DATA_BLOCK "G279M"
TITLE =DBG279M  HEATING KILN 1 + 2
//COPYRIGHT:    (C) 2009  BUHLER AG, CH-9240 UZWIL, SWITZERLAND
//
//PRODUCT:      WinCoS_BIW01_09
//
//TITLE:        HEATING KILN 1 + 2
//                Machine group DB
//                Maschinengruppen-DB
//
//-------------------------------------------------------------------------
//
//IDENT:        AUTHOR:             DEPT:             DATE:
//
//P01_DB379.1.0 K.Renz              CSB41             30.Sep.2009
//              1st Release
//
//-------------------------------------------------------------------------
//
//PURPOSE:
//
//MANUAL :
//
//RESTRICTIONS:
//
//-------------------------------------------------------------------------
AUTHOR : KR
FAMILY : USW
NAME : DBG279M
VERSION : 0.0

"G279M_Code"
BEGIN
   Gr.FcCode := 0;
   Gr.Spare2 := 0;
   Gr.Spare4 := 0;
   Gr.Spare6 := 0;
   Gr.OutEmptyingTime := 0;
   Gr.ChangeBit.spare := B#16#0;
   Gr.ChangeBit.CBit1 := FALSE;
   Gr.ChangeBit.CBit2 := FALSE;
   Gr.ChangeBit.CBit3 := FALSE;
   Gr.ChangeBit.CBit4 := FALSE;
   Gr.StCode := 0;
   Gr.InEnableGr := FALSE;
   Gr.CmdContinue := FALSE;
   Gr.CmdRestartIdling := FALSE;
   Gr.InReleaseEmptyingTime := FALSE;
   Gr.InFeeding := FALSE;
   Gr.InOutAutostartMan := FALSE;
   Gr.InPreStart := FALSE;
   Gr.CmdManualOff := FALSE;
   Gr.CmdOff := FALSE;
   Gr.CmdOn := FALSE;
   Gr.CmdNext := FALSE;
   Gr.CmdFaultReset := FALSE;
   Gr.InOccupied := FALSE;
   Gr.InManual := FALSE;
   Gr.InLoadedSec := FALSE;
   Gr.InSeqStop := FALSE;
   Gr.ModePassive := FALSE;
   Gr.ModeActive := FALSE;
   Gr.ModeIdling := FALSE;
   Gr.spare163 := FALSE;
   Gr.spare164 := FALSE;
   Gr.spare165 := FALSE;
   Gr.spare166 := FALSE;
   Gr.spare167 := FALSE;
   Gr.StStopped := FALSE;
   Gr.StStarting := FALSE;
   Gr.StStarted := FALSE;
   Gr.StStopping := FALSE;
   Gr.StFault := FALSE;
   Gr.OutLoaded := FALSE;
   Gr.OutWarning := FALSE;
   Gr.OutFeeding := FALSE;
   Gr.OutEnableEl := FALSE;
   Gr.OutEnable1 := FALSE;
   Gr.OutHWStop := FALSE;
   Gr.OutDPFault := FALSE;
   Gr.OutAutostart := FALSE;
   Gr.OutManual := FALSE;
   Gr.OutHornOn := FALSE;
   Gr.OutEnablePrevGr := FALSE;
   Gr.VarStopped := FALSE;
   Gr.VarStarted := FALSE;
   Gr.VarFault := FALSE;
   Gr.VarStartwarning := FALSE;
   Gr.VarFlag1s := FALSE;
   Gr.OutEmptyingTimeDone := FALSE;
   Gr.OutNewWay := FALSE;
   Gr.OutSeqStop := FALSE;
   Gr.OutIdlingTime := 0;
   Gr.InCodePreselect := 0;
   Gr.InLine := 0;
   Gr.InCode := 0;
   Gr.OutCode := 0;
   Gr.Par.ParObjectNo := 27900;
   Gr.Par.ParMgr := TRUE;
   Gr.Par.ParWgr := FALSE;
   Gr.Par.ParGgr := FALSE;
   Gr.Par.ParHornCode := 10;
   Gr.Par.ParIdling := 2;
   Gr.Par.ParEmptyingTime := 0;
   Gr.Par.Para1_0 := FALSE;
   Gr.Par.Para1_1 := FALSE;
   Gr.Par.Para1_2 := FALSE;
   Gr.Par.Para1_3 := FALSE;
   Gr.Par.Para1_4 := FALSE;
   Gr.Par.Para1_5 := FALSE;
   Gr.Par.Para1_6 := FALSE;
   Gr.Par.Para1_7 := FALSE;
   Gr.Par.Para1_8 := FALSE;
   Gr.Par.Para1_9 := FALSE;
   Gr.Par.Para1_10 := FALSE;
   Gr.Par.Para1_11 := FALSE;
   Gr.Par.Para1_12 := FALSE;
   Gr.Par.Para1_13 := FALSE;
   Gr.Par.Para1_14 := FALSE;
   Gr.Par.Para1_15 := FALSE;
   Gr.Par.Para2 := 0;
   Gr.Par.Para3 := 0;
   Gr.Par.Para4 := 0;
   Gr.Par.Para5 := 0;
   InOutValue1 := L#0;
   InOutValue2 := L#0;
   OutWayConflict := FALSE;
   OutSelectionOk := FALSE;
   CmdNewValue := FALSE;
   CmdNewJob := FALSE;
   OutCodeOK := FALSE;
   InEndOfJob := FALSE;
   staWayOk := FALSE;
   EdgeStartRelease := FALSE;
   USW8 := FALSE;
   USW9 := FALSE;
   USW10 := FALSE;
   _A_3191_BTE10_Active := FALSE;
   _A_3291_BTE10_Active := FALSE;
   USW13 := FALSE;
   USW14 := FALSE;
   USW15 := FALSE;
   A_3161_KCL11.StCode := 0;
   A_3161_KCL11.InMonTrue := FALSE;
   A_3161_KCL11.InMonFalse := FALSE;
   A_3161_KCL11.InPreAlarmTrue := FALSE;
   A_3161_KCL11.InPreAlarmFalse := FALSE;
   A_3161_KCL11.InStopTrueTime := FALSE;
   A_3161_KCL11.InStopFalseTime := FALSE;
   A_3161_KCL11.InpTrue := FALSE;
   A_3161_KCL11.InpFaultDev := FALSE;
   A_3161_KCL11.CmdRstTrueTime := FALSE;
   A_3161_KCL11.CmdRstFalseTime := FALSE;
   A_3161_KCL11.CmdRunTimeoutTime := FALSE;
   A_3161_KCL11.CmdFaultReset := FALSE;
   A_3161_KCL11.InLocal := FALSE;
   A_3161_KCL11.spare0305 := FALSE;
   A_3161_KCL11.InReport := FALSE;
   A_3161_KCL11.OutTimeoutTime := FALSE;
   A_3161_KCL11.InHWStop := FALSE;
   A_3161_KCL11.InDPFault := FALSE;
   A_3161_KCL11.OutPreAlarmTrue := FALSE;
   A_3161_KCL11.OutPreAlarmFalse := FALSE;
   A_3161_KCL11.OutFlagPos := FALSE;
   A_3161_KCL11.OutFlagNeg := FALSE;
   A_3161_KCL11.OutpFaultReset := FALSE;
   A_3161_KCL11.OutTrue := FALSE;
   A_3161_KCL11.StFalse := FALSE;
   A_3161_KCL11.StCtoTrue := FALSE;
   A_3161_KCL11.StTrue := FALSE;
   A_3161_KCL11.StCtoFalse := FALSE;
   A_3161_KCL11.StFault := FALSE;
   A_3161_KCL11.OutAlarmNrLog := 0;
   A_3161_KCL11.Par.ParObjectNo := 27901;
   A_3161_KCL11.Par.ParMsgType := 7154;
   A_3161_KCL11.Par.ParHornCode := 10;
   A_3161_KCL11.Par.ParLogOff := FALSE;
   A_3161_KCL11.Par.spare0401 := FALSE;
   A_3161_KCL11.Par.Par2WorkingCond := FALSE;
   A_3161_KCL11.Par.ParFaultRetry := FALSE;
   A_3161_KCL11.Par.ParBinLevel := FALSE;
   A_3161_KCL11.Par.ParDelayChange := 20;
   A_3161_KCL11.Par.ParDelayTrue := 10;
   A_3161_KCL11.Par.ParDelayFalse := 0;
   A_3161_KCL11.Par.ParTimeoutTrue := 0;
   A_3161_KCL11.Par.ParTimeoutFalse := 0;
   A_3161_KCL11.Par.OutMonTime := 0;
   A_3161_KCL11.Par.OutTransitionTime := 0;
   A_3161_KCL11.Par.OutMonTrue := FALSE;
   A_3161_KCL11.Par.OutMonFalse := FALSE;
   A_3161_KCL11.Par.OutFlagFaultDev := FALSE;
   A_3161_KCL11.Par.OutDelayTime := 0;
   A_3161_KCL11_EXT_ON.StCode := 0;
   A_3161_KCL11_EXT_ON.InEnable := FALSE;
   A_3161_KCL11_EXT_ON.spare0201 := FALSE;
   A_3161_KCL11_EXT_ON.InContinuous := FALSE;
   A_3161_KCL11_EXT_ON.spare0203 := FALSE;
   A_3161_KCL11_EXT_ON.spare0204 := FALSE;
   A_3161_KCL11_EXT_ON.spare0205 := FALSE;
   A_3161_KCL11_EXT_ON.InpRun := FALSE;
   A_3161_KCL11_EXT_ON.InpFaultDev := FALSE;
   A_3161_KCL11_EXT_ON.CmdOff := FALSE;
   A_3161_KCL11_EXT_ON.CmdOn := FALSE;
   A_3161_KCL11_EXT_ON.CmdNext := FALSE;
   A_3161_KCL11_EXT_ON.CmdFaultReset := FALSE;
   A_3161_KCL11_EXT_ON.InLocal := FALSE;
   A_3161_KCL11_EXT_ON.InManual := FALSE;
   A_3161_KCL11_EXT_ON.InReport := FALSE;
   A_3161_KCL11_EXT_ON.InSeqStop := FALSE;
   A_3161_KCL11_EXT_ON.InHWStop := FALSE;
   A_3161_KCL11_EXT_ON.InDPFault := FALSE;
   A_3161_KCL11_EXT_ON.OutIdling := FALSE;
   A_3161_KCL11_EXT_ON.OutWarning := FALSE;
   A_3161_KCL11_EXT_ON.spare0404 := FALSE;
   A_3161_KCL11_EXT_ON.spare0405 := FALSE;
   A_3161_KCL11_EXT_ON.OutpFaultReset := FALSE;
   A_3161_KCL11_EXT_ON.OutpRun := FALSE;
   A_3161_KCL11_EXT_ON.StStopped := FALSE;
   A_3161_KCL11_EXT_ON.StStarting := FALSE;
   A_3161_KCL11_EXT_ON.StStarted := FALSE;
   A_3161_KCL11_EXT_ON.spare0503 := FALSE;
   A_3161_KCL11_EXT_ON.StFault := FALSE;
   A_3161_KCL11_EXT_ON.StFalse := FALSE;
   A_3161_KCL11_EXT_ON.spare0506 := FALSE;
   A_3161_KCL11_EXT_ON.OutPausing := FALSE;
   A_3161_KCL11_EXT_ON.OutAlarmNrLog := 0;
   A_3161_KCL11_EXT_ON.Par.ParObjectNo := 27902;
   A_3161_KCL11_EXT_ON.Par.ParMsgType := 7002;
   A_3161_KCL11_EXT_ON.Par.ParHornCode := 0;
   A_3161_KCL11_EXT_ON.Par.ParLogOff := FALSE;
   A_3161_KCL11_EXT_ON.Par.ParManual := TRUE;
   A_3161_KCL11_EXT_ON.Par.ParContinuous := TRUE;
   A_3161_KCL11_EXT_ON.Par.ParPulse := FALSE;
   A_3161_KCL11_EXT_ON.Par.ParPulsing := FALSE;
   A_3161_KCL11_EXT_ON.Par.ParFilter := FALSE;
   A_3161_KCL11_EXT_ON.Par.ParOnTime := 10;
   A_3161_KCL11_EXT_ON.Par.ParOffTime := 0;
   A_3161_KCL11_EXT_ON.Par.ParIdlingTime := 0;
   A_3161_KCL11_EXT_ON.Par.ParDelayTime := 0;
   A_3161_KCL11_EXT_ON.Par.OutTime := 0;
   A_3161_KCL11_EXT_ON.Par.OutDelayTime := 0;
   A_3161_KCL11_EXT_ON.Par.spare26 := 0;
   A_3161_KCL11_EXT_ON.Par.spare28 := 0;
   A_3161_KCL11_EXT_ON.Par.InOutManPulseLen := 0;
   A_3161_KCL11_ON.StCode := 0;
   A_3161_KCL11_ON.InMonTrue := FALSE;
   A_3161_KCL11_ON.InMonFalse := FALSE;
   A_3161_KCL11_ON.InPreAlarmTrue := FALSE;
   A_3161_KCL11_ON.InPreAlarmFalse := FALSE;
   A_3161_KCL11_ON.InStopTrueTime := FALSE;
   A_3161_KCL11_ON.InStopFalseTime := FALSE;
   A_3161_KCL11_ON.InpTrue := FALSE;
   A_3161_KCL11_ON.InpFaultDev := FALSE;
   A_3161_KCL11_ON.CmdRstTrueTime := FALSE;
   A_3161_KCL11_ON.CmdRstFalseTime := FALSE;
   A_3161_KCL11_ON.CmdRunTimeoutTime := FALSE;
   A_3161_KCL11_ON.CmdFaultReset := FALSE;
   A_3161_KCL11_ON.InLocal := FALSE;
   A_3161_KCL11_ON.spare0305 := FALSE;
   A_3161_KCL11_ON.InReport := FALSE;
   A_3161_KCL11_ON.OutTimeoutTime := FALSE;
   A_3161_KCL11_ON.InHWStop := FALSE;
   A_3161_KCL11_ON.InDPFault := FALSE;
   A_3161_KCL11_ON.OutPreAlarmTrue := FALSE;
   A_3161_KCL11_ON.OutPreAlarmFalse := FALSE;
   A_3161_KCL11_ON.OutFlagPos := FALSE;
   A_3161_KCL11_ON.OutFlagNeg := FALSE;
   A_3161_KCL11_ON.OutpFaultReset := FALSE;
   A_3161_KCL11_ON.OutTrue := FALSE;
   A_3161_KCL11_ON.StFalse := FALSE;
   A_3161_KCL11_ON.StCtoTrue := FALSE;
   A_3161_KCL11_ON.StTrue := FALSE;
   A_3161_KCL11_ON.StCtoFalse := FALSE;
   A_3161_KCL11_ON.StFault := FALSE;
   A_3161_KCL11_ON.OutAlarmNrLog := 0;
   A_3161_KCL11_ON.Par.ParObjectNo := 27903;
   A_3161_KCL11_ON.Par.ParMsgType := 7154;
   A_3161_KCL11_ON.Par.ParHornCode := 0;
   A_3161_KCL11_ON.Par.ParLogOff := FALSE;
   A_3161_KCL11_ON.Par.spare0401 := FALSE;
   A_3161_KCL11_ON.Par.Par2WorkingCond := FALSE;
   A_3161_KCL11_ON.Par.ParFaultRetry := FALSE;
   A_3161_KCL11_ON.Par.ParBinLevel := FALSE;
   A_3161_KCL11_ON.Par.ParDelayChange := 20;
   A_3161_KCL11_ON.Par.ParDelayTrue := 10;
   A_3161_KCL11_ON.Par.ParDelayFalse := 0;
   A_3161_KCL11_ON.Par.ParTimeoutTrue := 0;
   A_3161_KCL11_ON.Par.ParTimeoutFalse := 0;
   A_3161_KCL11_ON.Par.OutMonTime := 0;
   A_3161_KCL11_ON.Par.OutTransitionTime := 0;
   A_3161_KCL11_ON.Par.OutMonTrue := FALSE;
   A_3161_KCL11_ON.Par.OutMonFalse := FALSE;
   A_3161_KCL11_ON.Par.OutFlagFaultDev := FALSE;
   A_3161_KCL11_ON.Par.OutDelayTime := 0;
   A_3161_KCL11_AI.StCode := 0;
   A_3161_KCL11_AI.InMonLL := FALSE;
   A_3161_KCL11_AI.InMonL := FALSE;
   A_3161_KCL11_AI.InMonMid := FALSE;
   A_3161_KCL11_AI.InMonH := FALSE;
   A_3161_KCL11_AI.InMonHH := FALSE;
   A_3161_KCL11_AI.spare0205 := FALSE;
   A_3161_KCL11_AI.InpFaultAI := FALSE;
   A_3161_KCL11_AI.InpFaultDev := FALSE;
   A_3161_KCL11_AI.InHWStop := FALSE;
   A_3161_KCL11_AI.InDPFault := FALSE;
   A_3161_KCL11_AI.InDisable := FALSE;
   A_3161_KCL11_AI.CmdFaultReset := FALSE;
   A_3161_KCL11_AI.InLocal := FALSE;
   A_3161_KCL11_AI.spare0305 := FALSE;
   A_3161_KCL11_AI.InReport := FALSE;
   A_3161_KCL11_AI.spare0307 := FALSE;
   A_3161_KCL11_AI.OutLL := FALSE;
   A_3161_KCL11_AI.OutL := FALSE;
   A_3161_KCL11_AI.OutH := FALSE;
   A_3161_KCL11_AI.OutHH := FALSE;
   A_3161_KCL11_AI.OutOverflow := FALSE;
   A_3161_KCL11_AI.spare0405 := FALSE;
   A_3161_KCL11_AI.OutFaultAI := FALSE;
   A_3161_KCL11_AI.spare0407 := FALSE;
   A_3161_KCL11_AI.StLL := FALSE;
   A_3161_KCL11_AI.StL := FALSE;
   A_3161_KCL11_AI.StMid := FALSE;
   A_3161_KCL11_AI.StH := FALSE;
   A_3161_KCL11_AI.StHH := FALSE;
   A_3161_KCL11_AI.StFaultAI := FALSE;
   A_3161_KCL11_AI.OutWarning := FALSE;
   A_3161_KCL11_AI.OutFaulted := FALSE;
   A_3161_KCL11_AI.InpValue := 0;
   A_3161_KCL11_AI.OutValuePc := 0;
   A_3161_KCL11_AI.OutValueUnits := L#0;
   A_3161_KCL11_AI.Msg.WarningDoneLL := FALSE;
   A_3161_KCL11_AI.Msg.WarningDoneL := FALSE;
   A_3161_KCL11_AI.Msg.WarningDoneMid := FALSE;
   A_3161_KCL11_AI.Msg.WarningDoneH := FALSE;
   A_3161_KCL11_AI.Msg.WarningDoneHH := FALSE;
   A_3161_KCL11_AI.Msg.FaultDoneLL := FALSE;
   A_3161_KCL11_AI.Msg.FaultDoneL := FALSE;
   A_3161_KCL11_AI.Msg.FaultDoneMid := FALSE;
   A_3161_KCL11_AI.Msg.FaultDoneH := FALSE;
   A_3161_KCL11_AI.Msg.FaultDoneHH := FALSE;
   A_3161_KCL11_AI.Msg.FaultDoneDev := FALSE;
   A_3161_KCL11_AI.Msg.FaultDoneAI := FALSE;
   A_3161_KCL11_AI.OutAlarmNrLog := 0;
   A_3161_KCL11_AI.Par.ParObjectNo := 27904;
   A_3161_KCL11_AI.Par.ParMsgType := 7252;
   A_3161_KCL11_AI.Par.ParHornCode := 10;
   A_3161_KCL11_AI.Par.ParLogOff := FALSE;
   A_3161_KCL11_AI.Par.ParSpare0401 := FALSE;
   A_3161_KCL11_AI.Par.ParValueByUser := FALSE;
   A_3161_KCL11_AI.Par.ParLimitsPc := TRUE;
   A_3161_KCL11_AI.Par.ParWago := FALSE;
   A_3161_KCL11_AI.Par.ParNoHornByWarning := FALSE;
   A_3161_KCL11_AI.Par.ParWarningLL := FALSE;
   A_3161_KCL11_AI.Par.ParWarningL := FALSE;
   A_3161_KCL11_AI.Par.ParWarningMid := FALSE;
   A_3161_KCL11_AI.Par.ParWarningH := FALSE;
   A_3161_KCL11_AI.Par.ParWarningHH := FALSE;
   A_3161_KCL11_AI.Par.ParPreAlarmLL := FALSE;
   A_3161_KCL11_AI.Par.ParPreAlarmL := FALSE;
   A_3161_KCL11_AI.Par.ParPreAlarmMid := FALSE;
   A_3161_KCL11_AI.Par.ParPreAlarmH := FALSE;
   A_3161_KCL11_AI.Par.ParPreAlarmHH := FALSE;
   A_3161_KCL11_AI.Par.ParUnitsByZeroDigit := L#0;
   A_3161_KCL11_AI.Par.ParUnitsByMaxDigit := L#16384;
   A_3161_KCL11_AI.Par.ParUnitsBy100Pc := L#10000;
   A_3161_KCL11_AI.Par.ParLimitLL := L#-1;
   A_3161_KCL11_AI.Par.ParLimitL := L#0;
   A_3161_KCL11_AI.Par.ParLimitH := L#7000;
   A_3161_KCL11_AI.Par.ParLimitHH := L#8000;
   A_3161_KCL11_AI.Par.ParMonTimeLL := 0;
   A_3161_KCL11_AI.Par.ParMonTimeL := 0;
   A_3161_KCL11_AI.Par.ParMonTimeMid := 0;
   A_3161_KCL11_AI.Par.ParMonTimeH := 0;
   A_3161_KCL11_AI.Par.ParMonTimeHH := 0;
   A_3161_KCL11_AI.Par.ParDelayTimeDown := 10;
   A_3161_KCL11_AI.Par.ParDelayTimeUp := 10;
   A_3161_KCL11_AI.Par.ParDelayTime := 30;
   A_3161_KCL11_AI.Par.OutMonTimeLL := 0;
   A_3161_KCL11_AI.Par.OutMonTimeL := 0;
   A_3161_KCL11_AI.Par.OutMonTimeMid := 0;
   A_3161_KCL11_AI.Par.OutMonTimeH := 0;
   A_3161_KCL11_AI.Par.OutMonTimeHH := 0;
   A_3161_KCL11_AI.Par.OutDelayTimeDown := 0;
   A_3161_KCL11_AI.Par.OutDelayTimeUp := 0;
   A_3161_KCL11_AI.Par.OutDelayTime := 0;
   A_3161_KCL11_AI.Par.Spare66 := 0;
   A_3161_KCL11_AO.StCode := 0;
   A_3161_KCL11_AO.InDisable := FALSE;
   A_3161_KCL11_AO.spare0201 := FALSE;
   A_3161_KCL11_AO.spare0202 := FALSE;
   A_3161_KCL11_AO.spare0203 := FALSE;
   A_3161_KCL11_AO.spare0204 := FALSE;
   A_3161_KCL11_AO.spare0205 := FALSE;
   A_3161_KCL11_AO.spare0206 := FALSE;
   A_3161_KCL11_AO.InpFaultDev := FALSE;
   A_3161_KCL11_AO.spare0300 := FALSE;
   A_3161_KCL11_AO.spare0301 := FALSE;
   A_3161_KCL11_AO.spare0302 := FALSE;
   A_3161_KCL11_AO.CmdFaultReset := FALSE;
   A_3161_KCL11_AO.InLocal := FALSE;
   A_3161_KCL11_AO.InManual := FALSE;
   A_3161_KCL11_AO.InReport := FALSE;
   A_3161_KCL11_AO.spare0307 := FALSE;
   A_3161_KCL11_AO.InHWStop := FALSE;
   A_3161_KCL11_AO.InDPFault := FALSE;
   A_3161_KCL11_AO.spare0402 := FALSE;
   A_3161_KCL11_AO.spare0403 := FALSE;
   A_3161_KCL11_AO.spare0404 := FALSE;
   A_3161_KCL11_AO.OutpFaultReset := FALSE;
   A_3161_KCL11_AO.OutMin := FALSE;
   A_3161_KCL11_AO.OutMax := FALSE;
   A_3161_KCL11_AO.StOff := FALSE;
   A_3161_KCL11_AO.spare0501 := FALSE;
   A_3161_KCL11_AO.StOn := FALSE;
   A_3161_KCL11_AO.spare0503 := FALSE;
   A_3161_KCL11_AO.StFault := FALSE;
   A_3161_KCL11_AO.OutpValue := 0;
   A_3161_KCL11_AO.InOutValuePc := 0;
   A_3161_KCL11_AO.InOutValueUnits := L#0;
   A_3161_KCL11_AO.ASW := L#0;
   A_3161_KCL11_AO.OutAlarmNrLog := 0;
   A_3161_KCL11_AO.Par.ParObjectNo := 27905;
   A_3161_KCL11_AO.Par.ParMsgType := 7241;
   A_3161_KCL11_AO.Par.ParHornCode := 10;
   A_3161_KCL11_AO.Par.ParLogOff := FALSE;
   A_3161_KCL11_AO.Par.ParFU := FALSE;
   A_3161_KCL11_AO.Par.ParValuePc := TRUE;
   A_3161_KCL11_AO.Par.ParLimitsPc := TRUE;
   A_3161_KCL11_AO.Par.ParWago := FALSE;
   A_3161_KCL11_AO.Par.ParUnitsByZeroDigit := L#0;
   A_3161_KCL11_AO.Par.ParUnitsByMaxDigit := L#16875;
   A_3161_KCL11_AO.Par.ParUnitsBy100Pc := L#10000;
   A_3161_KCL11_AO.Par.ParLimitMin := L#0;
   A_3161_KCL11_AO.Par.ParLimitMax := L#27648;
   A_3161_KCL11_AO.Par.ParDelayTime := 30;
   A_3161_KCL11_AO.Par.OutDelayTime := 0;
   A_3161_KCL11_REG_ON.StCode := 0;
   A_3161_KCL11_REG_ON.InMonTrue := FALSE;
   A_3161_KCL11_REG_ON.InMonFalse := FALSE;
   A_3161_KCL11_REG_ON.InPreAlarmTrue := FALSE;
   A_3161_KCL11_REG_ON.InPreAlarmFalse := FALSE;
   A_3161_KCL11_REG_ON.InStopTrueTime := FALSE;
   A_3161_KCL11_REG_ON.InStopFalseTime := FALSE;
   A_3161_KCL11_REG_ON.InpTrue := FALSE;
   A_3161_KCL11_REG_ON.InpFaultDev := FALSE;
   A_3161_KCL11_REG_ON.CmdRstTrueTime := FALSE;
   A_3161_KCL11_REG_ON.CmdRstFalseTime := FALSE;
   A_3161_KCL11_REG_ON.CmdRunTimeoutTime := FALSE;
   A_3161_KCL11_REG_ON.CmdFaultReset := FALSE;
   A_3161_KCL11_REG_ON.InLocal := FALSE;
   A_3161_KCL11_REG_ON.spare0305 := FALSE;
   A_3161_KCL11_REG_ON.InReport := FALSE;
   A_3161_KCL11_REG_ON.OutTimeoutTime := FALSE;
   A_3161_KCL11_REG_ON.InHWStop := FALSE;
   A_3161_KCL11_REG_ON.InDPFault := FALSE;
   A_3161_KCL11_REG_ON.OutPreAlarmTrue := FALSE;
   A_3161_KCL11_REG_ON.OutPreAlarmFalse := FALSE;
   A_3161_KCL11_REG_ON.OutFlagPos := FALSE;
   A_3161_KCL11_REG_ON.OutFlagNeg := FALSE;
   A_3161_KCL11_REG_ON.OutpFaultReset := FALSE;
   A_3161_KCL11_REG_ON.OutTrue := FALSE;
   A_3161_KCL11_REG_ON.StFalse := FALSE;
   A_3161_KCL11_REG_ON.StCtoTrue := FALSE;
   A_3161_KCL11_REG_ON.StTrue := FALSE;
   A_3161_KCL11_REG_ON.StCtoFalse := FALSE;
   A_3161_KCL11_REG_ON.StFault := FALSE;
   A_3161_KCL11_REG_ON.OutAlarmNrLog := 0;
   A_3161_KCL11_REG_ON.Par.ParObjectNo := 27906;
   A_3161_KCL11_REG_ON.Par.ParMsgType := 7154;
   A_3161_KCL11_REG_ON.Par.ParHornCode := 10;
   A_3161_KCL11_REG_ON.Par.ParLogOff := FALSE;
   A_3161_KCL11_REG_ON.Par.spare0401 := FALSE;
   A_3161_KCL11_REG_ON.Par.Par2WorkingCond := FALSE;
   A_3161_KCL11_REG_ON.Par.ParFaultRetry := FALSE;
   A_3161_KCL11_REG_ON.Par.ParBinLevel := FALSE;
   A_3161_KCL11_REG_ON.Par.ParDelayChange := 20;
   A_3161_KCL11_REG_ON.Par.ParDelayTrue := 10;
   A_3161_KCL11_REG_ON.Par.ParDelayFalse := 0;
   A_3161_KCL11_REG_ON.Par.ParTimeoutTrue := 0;
   A_3161_KCL11_REG_ON.Par.ParTimeoutFalse := 0;
   A_3161_KCL11_REG_ON.Par.OutMonTime := 0;
   A_3161_KCL11_REG_ON.Par.OutTransitionTime := 0;
   A_3161_KCL11_REG_ON.Par.OutMonTrue := FALSE;
   A_3161_KCL11_REG_ON.Par.OutMonFalse := FALSE;
   A_3161_KCL11_REG_ON.Par.OutFlagFaultDev := FALSE;
   A_3161_KCL11_REG_ON.Par.OutDelayTime := 0;
   A_3161_KCL11_REM_OP.StCode := 0;
   A_3161_KCL11_REM_OP.InMonTrue := FALSE;
   A_3161_KCL11_REM_OP.InMonFalse := FALSE;
   A_3161_KCL11_REM_OP.InPreAlarmTrue := FALSE;
   A_3161_KCL11_REM_OP.InPreAlarmFalse := FALSE;
   A_3161_KCL11_REM_OP.InStopTrueTime := FALSE;
   A_3161_KCL11_REM_OP.InStopFalseTime := FALSE;
   A_3161_KCL11_REM_OP.InpTrue := FALSE;
   A_3161_KCL11_REM_OP.InpFaultDev := FALSE;
   A_3161_KCL11_REM_OP.CmdRstTrueTime := FALSE;
   A_3161_KCL11_REM_OP.CmdRstFalseTime := FALSE;
   A_3161_KCL11_REM_OP.CmdRunTimeoutTime := FALSE;
   A_3161_KCL11_REM_OP.CmdFaultReset := FALSE;
   A_3161_KCL11_REM_OP.InLocal := FALSE;
   A_3161_KCL11_REM_OP.spare0305 := FALSE;
   A_3161_KCL11_REM_OP.InReport := FALSE;
   A_3161_KCL11_REM_OP.OutTimeoutTime := FALSE;
   A_3161_KCL11_REM_OP.InHWStop := FALSE;
   A_3161_KCL11_REM_OP.InDPFault := FALSE;
   A_3161_KCL11_REM_OP.OutPreAlarmTrue := FALSE;
   A_3161_KCL11_REM_OP.OutPreAlarmFalse := FALSE;
   A_3161_KCL11_REM_OP.OutFlagPos := FALSE;
   A_3161_KCL11_REM_OP.OutFlagNeg := FALSE;
   A_3161_KCL11_REM_OP.OutpFaultReset := FALSE;
   A_3161_KCL11_REM_OP.OutTrue := FALSE;
   A_3161_KCL11_REM_OP.StFalse := FALSE;
   A_3161_KCL11_REM_OP.StCtoTrue := FALSE;
   A_3161_KCL11_REM_OP.StTrue := FALSE;
   A_3161_KCL11_REM_OP.StCtoFalse := FALSE;
   A_3161_KCL11_REM_OP.StFault := FALSE;
   A_3161_KCL11_REM_OP.OutAlarmNrLog := 0;
   A_3161_KCL11_REM_OP.Par.ParObjectNo := 27907;
   A_3161_KCL11_REM_OP.Par.ParMsgType := 7154;
   A_3161_KCL11_REM_OP.Par.ParHornCode := 10;
   A_3161_KCL11_REM_OP.Par.ParLogOff := FALSE;
   A_3161_KCL11_REM_OP.Par.spare0401 := FALSE;
   A_3161_KCL11_REM_OP.Par.Par2WorkingCond := FALSE;
   A_3161_KCL11_REM_OP.Par.ParFaultRetry := FALSE;
   A_3161_KCL11_REM_OP.Par.ParBinLevel := FALSE;
   A_3161_KCL11_REM_OP.Par.ParDelayChange := 20;
   A_3161_KCL11_REM_OP.Par.ParDelayTrue := 10;
   A_3161_KCL11_REM_OP.Par.ParDelayFalse := 0;
   A_3161_KCL11_REM_OP.Par.ParTimeoutTrue := 0;
   A_3161_KCL11_REM_OP.Par.ParTimeoutFalse := 0;
   A_3161_KCL11_REM_OP.Par.OutMonTime := 0;
   A_3161_KCL11_REM_OP.Par.OutTransitionTime := 0;
   A_3161_KCL11_REM_OP.Par.OutMonTrue := FALSE;
   A_3161_KCL11_REM_OP.Par.OutMonFalse := FALSE;
   A_3161_KCL11_REM_OP.Par.OutFlagFaultDev := FALSE;
   A_3161_KCL11_REM_OP.Par.OutDelayTime := 0;
   A_3161_KCL11_RUN.StCode := 0;
   A_3161_KCL11_RUN.InEnable := FALSE;
   A_3161_KCL11_RUN.spare0201 := FALSE;
   A_3161_KCL11_RUN.InContinuous := FALSE;
   A_3161_KCL11_RUN.spare0203 := FALSE;
   A_3161_KCL11_RUN.spare0204 := FALSE;
   A_3161_KCL11_RUN.spare0205 := FALSE;
   A_3161_KCL11_RUN.InpRun := FALSE;
   A_3161_KCL11_RUN.InpFaultDev := FALSE;
   A_3161_KCL11_RUN.CmdOff := FALSE;
   A_3161_KCL11_RUN.CmdOn := FALSE;
   A_3161_KCL11_RUN.CmdNext := FALSE;
   A_3161_KCL11_RUN.CmdFaultReset := FALSE;
   A_3161_KCL11_RUN.InLocal := FALSE;
   A_3161_KCL11_RUN.InManual := FALSE;
   A_3161_KCL11_RUN.InReport := FALSE;
   A_3161_KCL11_RUN.InSeqStop := FALSE;
   A_3161_KCL11_RUN.InHWStop := FALSE;
   A_3161_KCL11_RUN.InDPFault := FALSE;
   A_3161_KCL11_RUN.OutIdling := FALSE;
   A_3161_KCL11_RUN.OutWarning := FALSE;
   A_3161_KCL11_RUN.spare0404 := FALSE;
   A_3161_KCL11_RUN.spare0405 := FALSE;
   A_3161_KCL11_RUN.OutpFaultReset := FALSE;
   A_3161_KCL11_RUN.OutpRun := FALSE;
   A_3161_KCL11_RUN.StStopped := FALSE;
   A_3161_KCL11_RUN.StStarting := FALSE;
   A_3161_KCL11_RUN.StStarted := FALSE;
   A_3161_KCL11_RUN.spare0503 := FALSE;
   A_3161_KCL11_RUN.StFault := FALSE;
   A_3161_KCL11_RUN.StFalse := FALSE;
   A_3161_KCL11_RUN.spare0506 := FALSE;
   A_3161_KCL11_RUN.OutPausing := FALSE;
   A_3161_KCL11_RUN.OutAlarmNrLog := 0;
   A_3161_KCL11_RUN.Par.ParObjectNo := 27908;
   A_3161_KCL11_RUN.Par.ParMsgType := 7002;
   A_3161_KCL11_RUN.Par.ParHornCode := 0;
   A_3161_KCL11_RUN.Par.ParLogOff := FALSE;
   A_3161_KCL11_RUN.Par.ParManual := TRUE;
   A_3161_KCL11_RUN.Par.ParContinuous := TRUE;
   A_3161_KCL11_RUN.Par.ParPulse := FALSE;
   A_3161_KCL11_RUN.Par.ParPulsing := FALSE;
   A_3161_KCL11_RUN.Par.ParFilter := FALSE;
   A_3161_KCL11_RUN.Par.ParOnTime := 10;
   A_3161_KCL11_RUN.Par.ParOffTime := 0;
   A_3161_KCL11_RUN.Par.ParIdlingTime := 0;
   A_3161_KCL11_RUN.Par.ParDelayTime := 0;
   A_3161_KCL11_RUN.Par.OutTime := 0;
   A_3161_KCL11_RUN.Par.OutDelayTime := 0;
   A_3161_KCL11_RUN.Par.spare26 := 0;
   A_3161_KCL11_RUN.Par.spare28 := 0;
   A_3161_KCL11_RUN.Par.InOutManPulseLen := 0;
END_DATA_BLOCK

